// TwinCAT 3 PLC project HMI
// ProgramVersion: 3.1.4023.0
// libraries:
//   Tc2_Standard, * (Beckhoff Automation GmbH)
//   Tc2_System, * (Beckhoff Automation GmbH)
//   Tc3_Module, * (Beckhoff Automation GmbH)
//   VisuSymbols,3.5.10.0,System
// project tree:
//   / GlobalTextList.TcGTLO, PlcTask.TcTTO, Visualization Manager.TcVMO (not stored)
//   POUs/ MAIN.TcPOU
//   VISUs/ STN500HMI.TcVIS, STNX00HMI.TcVIS, STN400HMI.TcVIS
// real-time tasks:
//   TASK PlcTask: cycle T#10ms, priority 20, ADS port 350
//   TASK PlcTask1: cycle T#10ms, priority 21, ADS port 351

CONFIGURATION HMI
    RESOURCE PLC ON TwinCAT3
        TASK PlcTask(INTERVAL := T#10ms, PRIORITY := 21);
        PROGRAM MAIN WITH PlcTask : MAIN;
    END_RESOURCE
END_CONFIGURATION

// ---- POUs/MAIN.TcPOU
PROGRAM MAIN
VAR
END_VAR

END_PROGRAM

// ---- GlobalTextList.TcGTLO
TEXTLIST GlobalTextList
  972 = 'Auto'
  720 = 'Auto Mode'
  224 = 'Auto mode'
  867 = 'Auto-Mode'
  571 = 'Emergency'
  133 = 'Full-Auto'
  759 = 'Gate Open'
  612 = 'Go Home'
  464 = 'Go To storage'
  668 = 'j'
  822 = 'Label'
  754 = 'Leave'
  393 = 'Line'
  219 = 'Low Soeed'
  3 = 'Low Speed'
  692 = 'Man.'
  879 = 'Manual'
  696 = 'Mode'
  644 = 'MOde'
  816 = 'Pause'
  818 = 'Pause Auto'
  450 = 'Paused'
  446 = 'Pick'
  947 = 'Run'
  896 = 'Rush Order'
  701 = 'Rush Production'
  186 = 'Semi-Auto'
  705 = 'Start Auto'
  268 = 'STN100'
  855 = 'STN200'
  275 = 'STN300'
  739 = 'STN400'
  581 = 'STN500'
  975 = 'Stop Auto'
  553 = 'Stoppe'
  239 = 'Stopped'
  266 = 'ToHome'
  507 = 'ToSensor'
  373 = 'ToStorage'
  130 = 'ToTable'
END_TEXTLIST

// ---- VISUs/STN500HMI.TcVIS
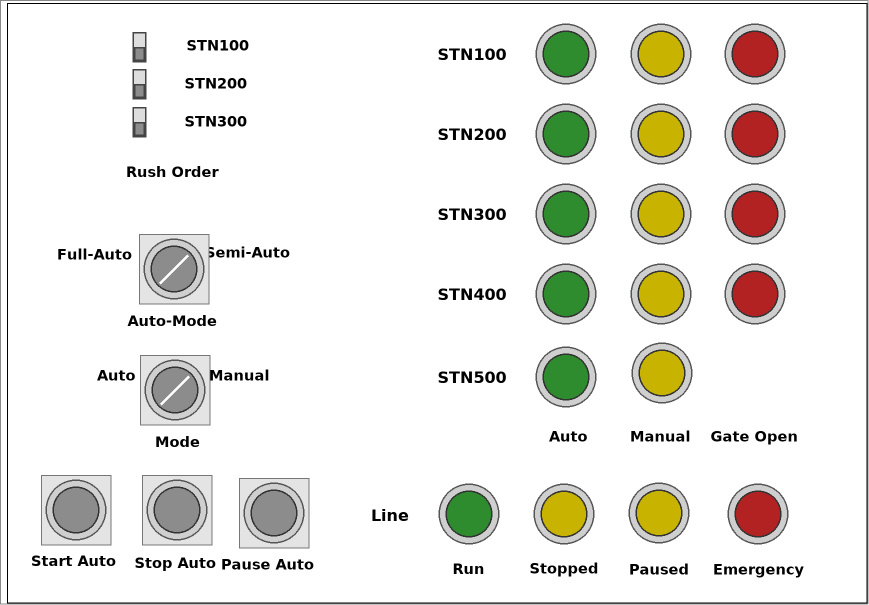
VISUALIZATION STN500HMI  // 869x605
    RoundedRectangle (7,3 860x600)
    RotarySwitch (140,355 70x70), behaviour: TOGGLE, style: Switch-RotarySwitch-Gray
    Label (93,359 47x33), "Auto"
    Label (151,427 53x30), "Mode"
    Label (203,360 73x31), "Manual"
    Label (202,239 91x27), "Semi-Auto"
    RotarySwitch (139,234 70x70), behaviour: TOGGLE, style: Switch-RotarySwitch-Gray
    Label (50,238 89x33), "Full-Auto"
    Label (121,305 103x32), "Auto-Mode"
    DipSwitch (102,107 75x30), behaviour: TOGGLE, style: Switch-DipSwitch-Gray
    DipSwitch (102,69 75x30), behaviour: TOGGLE, style: Switch-DipSwitch-Gray
    DipSwitch (102,32 75x30), behaviour: TOGGLE, style: Switch-DipSwitch-Gray
    Label (91,157 163x30), "Rush Order"
    Label (182,30 72x31), "STN100"
    Label (180,64 72x39), "STN200"
    Label (180,106 72x31), "STN300"
    Label (427,34 90x41), "STN100"
    Label (427,114 90x41), "STN200"
    Label (427,194 90x41), "STN300"
    Label (427,274 90x41), "STN400"
    Label (427,357 90x41), "STN500"
    Lamp1 (531,19 70x70), style: Lamp-Lamp1-Green
    Lamp1 (531,99 70x70), style: Lamp-Lamp1-Green
    Lamp1 (531,179 70x70), style: Lamp-Lamp1-Green
    Lamp1 (531,259 70x70), style: Lamp-Lamp1-Green
    Lamp1 (531,342 70x70), style: Lamp-Lamp1-Green
    Lamp1 (626,19 70x70), style: Lamp-Lamp1-Yellow
    Lamp1 (626,99 70x70), style: Lamp-Lamp1-Yellow
    Lamp1 (626,179 70x70), style: Lamp-Lamp1-Yellow
    Lamp1 (626,259 70x70), style: Lamp-Lamp1-Yellow
    Lamp1 (720,19 70x70), style: Lamp-Lamp1-Red
    Lamp1 (720,99 70x70), style: Lamp-Lamp1-Red
    Lamp1 (720,179 70x70), style: Lamp-Lamp1-Red
    Lamp1 (720,259 70x70), style: Lamp-Lamp1-Red
    Label (545,420 47x33), "Auto"
    Label (615,415 91x43), "Manual"
    Label (709,415 91x43), "Gate Open"
    Lamp1 (627,338 70x70), style: Lamp-Lamp1-Yellow
    PushSwitch (41,475 70x70), behaviour: TOGGLE, style: Switch-PushSwitch-Gray
    PushSwitch (142,475 70x70), behaviour: TOGGLE, style: Switch-PushSwitch-Gray
    PushSwitch (239,478 70x70), behaviour: TOGGLE, style: Switch-PushSwitch-Gray
    Label (31,544 85x34), "Start Auto"
    Label (133,546 85x34), "Stop Auto"
    Label (219,546 97x37), "Pause Auto"
    Label (345,495 90x41), "Line"
    Lamp1 (434,479 70x70), style: Lamp-Lamp1-Green
    Lamp1 (529,479 70x70), style: Lamp-Lamp1-Yellow
    Lamp1 (723,479 70x70), style: Lamp-Lamp1-Red
    Label (713,548 91x43), "Emergency"
    Lamp1 (624,478 70x70), style: Lamp-Lamp1-Yellow
    Label (442,554 53x30), "Run"
    Label (523,555 82x27), "Stopped"
    Label (618,556 82x27), "Paused"
END_VISUALIZATION

// ---- VISUs/STNX00HMI.TcVIS
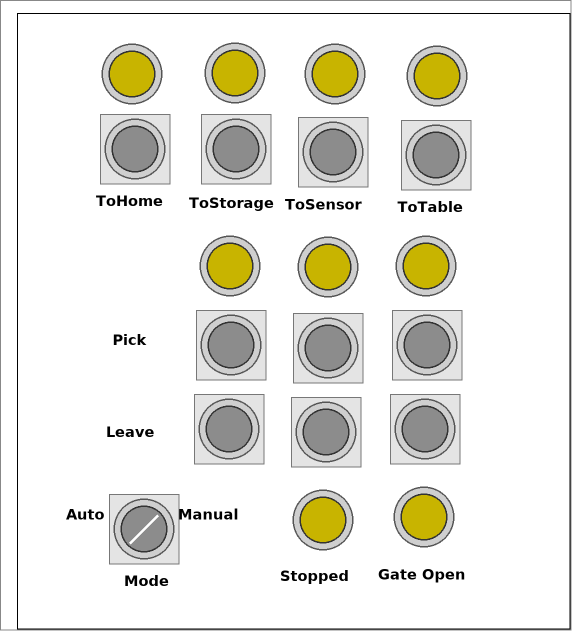
VISUALIZATION STNX00HMI  // 572x631
    RoundedRectangle (17,13 553x616)
    Label (62,498 47x33), "Auto"
    RotarySwitch (109,494 70x70), behaviour: TOGGLE, style: Switch-RotarySwitch-Gray
    Label (120,566 53x30), "Mode"
    Label (172,499 73x31), "Manual"
    PushSwitch (100,114 70x70), behaviour: TOGGLE, style: Switch-PushSwitch-Gray
    PushSwitch (201,114 70x70), behaviour: TOGGLE, style: Switch-PushSwitch-Gray
    PushSwitch (298,117 70x70), behaviour: TOGGLE, style: Switch-PushSwitch-Gray
    Label (87,184 85x34), "ToHome"
    Label (189,186 85x34), "ToStorage"
    Label (275,186 97x37), "ToSensor"
    PushSwitch (196,310 70x70), behaviour: TOGGLE, style: Switch-PushSwitch-Gray
    PushSwitch (293,313 70x70), behaviour: TOGGLE, style: Switch-PushSwitch-Gray
    Label (87,323 85x34), "Pick"
    PushSwitch (401,120 70x70), behaviour: TOGGLE, style: Switch-PushSwitch-Gray
    Label (388,190 85x34), "ToTable"
    Lamp1 (97,39 70x70), style: Lamp-Lamp1-Yellow
    Lamp1 (200,38 70x70), style: Lamp-Lamp1-Yellow
    Lamp1 (300,39 70x70), style: Lamp-Lamp1-Yellow
    Lamp1 (402,41 70x70), style: Lamp-Lamp1-Yellow
    Lamp1 (195,231 70x70), style: Lamp-Lamp1-Yellow
    Lamp1 (293,232 70x70), style: Lamp-Lamp1-Yellow
    Lamp1 (391,231 70x70), style: Lamp-Lamp1-Yellow
    PushSwitch (392,310 70x70), behaviour: TOGGLE, style: Switch-PushSwitch-Gray
    PushSwitch (194,394 70x70), behaviour: TOGGLE, style: Switch-PushSwitch-Gray
    PushSwitch (291,397 70x70), behaviour: TOGGLE, style: Switch-PushSwitch-Gray
    PushSwitch (390,394 70x70), behaviour: TOGGLE, style: Switch-PushSwitch-Gray
    Label (88,415 85x34), "Leave"
    Lamp1 (288,485 70x70), style: Lamp-Lamp1-Yellow
    Lamp1 (389,482 70x70), style: Lamp-Lamp1-Yellow
    Label (373,553 98x43), "Gate Open"
    Label (267,559 95x34), "Stopped"
END_VISUALIZATION

// ---- VISUs/STN400HMI.TcVIS
VISUALIZATION STN400HMI  // 2x2
END_VISUALIZATION
